SUBAPPLICATION Uebung_007a3_AX (* Blinker mit E_CYCLE, E_SWITCH und E_SR *)
  (* Standard: 61499-2; Description: Copyright (c) 2023 Meisterschulen am Ostbahnhof This program and the accompanying materials are made available under the terms of the Eclipse Public License 2.0 which is available at https://www.eclipse.org/legal/epl-2.0/ SPDX-License-Identifier: EPL-2.0 *)
  (* Version 1.0, 2023-10-23, Franz Höpfinger, Meisterschulen am Ostbahnhof, initial API and implementation and/or initial documentation *)
  PACKAGE Uebungen;
  IMPORT logiBUS::io::DI::logiBUS_DI::Input_I1;
  IMPORT logiBUS::io::DI::logiBUS_DI::Input_I2;
  IMPORT logiBUS::io::DI::logiBUS_DI_Events::BUTTON_SINGLE_CLICK;
  IMPORT logiBUS::io::DQ::logiBUS_DO::Output_Q1;
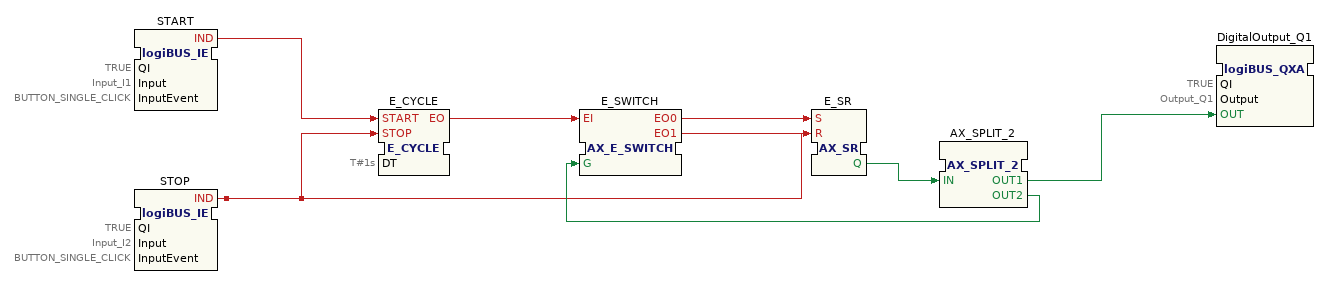
  (* Vorteil: dieser Blinker bleibt immer auf AUS stehen *)
  FBS
    DigitalOutput_Q1 : logiBUS::io::DQ::logiBUS_QXA(QI := TRUE, Output := Output_Q1);
    E_CYCLE : iec61499::events::E_CYCLE(DT := T#1s);
    START : logiBUS::io::DI::logiBUS_IE(QI := TRUE, Input := Input_I1, InputEvent := BUTTON_SINGLE_CLICK);
    STOP : logiBUS::io::DI::logiBUS_IE(QI := TRUE, Input := Input_I2, InputEvent := BUTTON_SINGLE_CLICK);
    E_SR : adapter::events::unidirectional::AX_SR;
    AX_SPLIT_2 : adapter::events::unidirectional::AX_SPLIT_2;
    E_SWITCH : adapter::events::unidirectional::AX_E_SWITCH;
  END_FBS
  EVENT_CONNECTIONS
    START.IND TO E_CYCLE.START;
    STOP.IND TO E_CYCLE.STOP;
    E_SWITCH.EO0 TO E_SR.S;
    E_SWITCH.EO1 TO E_SR.R;
    E_CYCLE.EO TO E_SWITCH.EI;
    STOP.IND TO E_SR.R;
  END_CONNECTIONS
  ADAPTER_CONNECTIONS
    E_SR.Q TO AX_SPLIT_2.IN;
    AX_SPLIT_2.OUT1 TO DigitalOutput_Q1.OUT;
    AX_SPLIT_2.OUT2 TO E_SWITCH.G;
  END_CONNECTIONS
END_SUBAPPLICATION
